FUNCTION_BLOCK BloqueioAtivaDesativa_HMI (* Service Interface Function Block Type *)
  (* Standard: 61499-2 *)
  (* Version 0.0, 02/03/2026, template *)
  PACKAGE Hidryco.HidrycoLib;
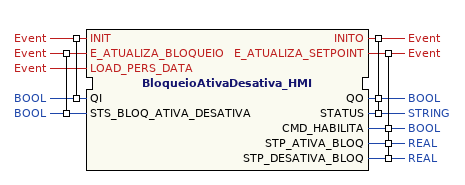
  EVENT_INPUT
    INIT WITH QI;
    E_ATUALIZA_BLOQUEIO WITH STS_BLOQ_ATIVA_DESATIVA;
    LOAD_PERS_DATA;
  END_EVENT
  EVENT_OUTPUT
    INITO WITH QO, STATUS;
    E_ATUALIZA_SETPOINT WITH CMD_HABILITA, STP_ATIVA_BLOQ, STP_DESATIVA_BLOQ;
  END_EVENT
  VAR_INPUT
    QI : BOOL;
    STS_BLOQ_ATIVA_DESATIVA : BOOL;
  END_VAR
  VAR_OUTPUT
    QO : BOOL; (* Event Output Qualifier *)
    STATUS : STRING; (* Service Status *)
    CMD_HABILITA : BOOL;
    STP_ATIVA_BLOQ : REAL;
    STP_DESATIVA_BLOQ : REAL;
  END_VAR
  SERVICE /
    SEQUENCE 
    END_SEQUENCE
  END_SERVICE
END_FUNCTION_BLOCK
